// TwinCAT 3 PLC project PLC
// Title: NotificationExample
// Company: Red Rock Controls Limited
// Author: Roger Christopher
// ProjectVersion: 1.0.1.0
// ProgramVersion: 3.1.4024.12
// libraries:
//   Tc2_Standard, * (Beckhoff Automation GmbH)
//   Tc2_System, * (Beckhoff Automation GmbH)
//   Tc3_Module, * (Beckhoff Automation GmbH)
//   tcl_BaseClasses, * (Red Rock Controls Limited)
// project tree:
//   GVLs/ Notifications.TcGVL
//   / PlcTask.TcTTO, PlcTask2.TcTTO
//   POUs/ MAIN_Task1.TcPOU, MAIN_Task2.TcPOU, T_MachineSettingsServer.TcPOU, T_MachineSettingsClient.TcPOU
//   Version/ Global_Version.TcGVL
// real-time tasks:
//   TASK PlcTask1: cycle T#1ms, priority 4, ADS port 350
//   TASK PlcTask2: cycle T#1ms, priority 5, ADS port 351

CONFIGURATION PLC
    RESOURCE PLC ON TwinCAT3
        TASK PlcTask(INTERVAL := T#1ms, PRIORITY := 4);
        TASK PlcTask2(INTERVAL := T#1ms, PRIORITY := 5);
        PROGRAM MAIN_Task1 WITH PlcTask : MAIN_Task1;
        PROGRAM MAIN_Task2 WITH PlcTask2 : MAIN_Task2;
    END_RESOURCE
END_CONFIGURATION

// ---- GVLs/Notifications.TcGVL
{attribute 'qualified_only'}
VAR_GLOBAL
	MachineSettingsLoaded  : T_Notification;
	MachineSettingsUpdated : T_Notification;
END_VAR

// ---- Version/Global_Version.TcGVL
{attribute 'TcGenerated'}
{attribute 'no-analysis'}
{attribute 'linkalways'}
// This function has been automatically generated from the project information.
VAR_GLOBAL CONSTANT
	{attribute 'const_non_replaced'}
	stLibVersion_NotificationExample : ST_LibVersion := (iMajor := 1, iMinor := 0, iBuild := 1, iRevision := 0, nFlags := 0, sVersion := '1.0.1.0');
END_VAR

// ---- POUs/MAIN_Task1.TcPOU
PROGRAM MAIN_Task1
VAR
    MachineSettingsServer : T_MachineSettingsServer; // Sends settings and loaded status to MachineSettingsClient running in separate context (task)
    Init            : BOOL := TRUE;

END_VAR

IF Init THEN
    // Manually resize the args buffer, as resizing 10,000 times produces a very long scan...
    Notifications.MachineSettingsUpdated.Args.Init(StreamLength := 60000);

    // Link the handler to the notification...
    Notifications.MachineSettingsLoaded
        .ClearNotificationHandlers()
    	.AddNotificationHandler(MAIN_Task2.MachineSettingsClient.OnSettingsLoaded);

    Notifications.MachineSettingsUpdated
        .ClearNotificationHandlers()
    	.AddNotificationHandler(MAIN_Task2.MachineSettingsClient.OnSettingsUpdated);

    Init := FALSE;
END_IF

// Run the server...
MachineSettingsServer.CyclicUpdate();

END_PROGRAM

// ---- POUs/T_MachineSettingsServer.TcPOU
FUNCTION_BLOCK T_MachineSettingsServer
VAR
    SettingsLoaded  : BOOL; // raises MachineSettingsLoaded notification, handled by T_MachineSettingsClient
    SettingsUpdated : BOOL; // raises MachoneSettingsUpdated notification, handled by T_MachineSettingsClient

    Settings : ARRAY[1..10000] OF UDINT;

END_VAR

METHOD CyclicUpdate
VAR_INST
    Init     : BOOL := TRUE;
    i        : UDINT;
    SendOnce : BOOL := TRUE; // set true to send single notifications
END_VAR
IF Init THEN
    // clear the flag...
    Init := FALSE;

    // write some values into the settings...
    FOR i := 1 TO 10000 DO
        Settings[i] := i;
    END_FOR
END_IF

IF SettingsLoaded THEN // manually set this flag to send SettingsLoaded notifications...
    IF SendOnce THEN // Set SendOnce to FALSE to send notification every scan - should still work if tasks run on separate isolated cores!
        SettingsLoaded := FALSE; 
    END_IF

    // raise the simple notification with no args...
    Notifications.MachineSettingsLoaded.Raise();
END_IF

IF SettingsUpdated THEN // manually set this flag to send SettingsUpdated notifications...
    IF SendOnce THEN // Set SendOnce to FALSE to send notification every scan - should still work if tasks run on separate isolated cores!
        SettingsUpdated := FALSE; 
    END_IF

    // write the seettings into the notification args...
    FOR i := 1 TO 10000 DO
        Notifications.MachineSettingsUpdated.Args.Add_UDINT(Settings[i]);
    END_FOR

    // raise the notification...
    Notifications.MachineSettingsUpdated.Raise();
END_IF
END_METHOD

END_FUNCTION_BLOCK

// ---- POUs/MAIN_Task2.TcPOU
PROGRAM MAIN_Task2
VAR
	MachineSettingsClient : T_MachineSettingsClient; // Receives settings and loaded status from MachineSettingsServer running in separate context (task)
END_VAR

MachineSettingsClient.HandleNotifications();

END_PROGRAM

// ---- POUs/T_MachineSettingsClient.TcPOU
FUNCTION_BLOCK T_MachineSettingsClient // Handles notifications of settings loaded and settings updated
VAR
    OnSettingsLoaded  : T_NotificationHandler;
    OnSettingsUpdated : T_NotificationHandler;

    SettingsLoadedCount : UDINT;
    LocalSettings       : ARRAY[1..10000] OF UDINT;
END_VAR

METHOD HandleNotifications
VAR
    i                   : UDINT;
END_VAR
IF OnSettingsLoaded.IsRaised() THEN
    // do something...
    SettingsLoadedCount := SettingsLoadedCount + 1;
END_IF

IF OnSettingsUpdated.IsRaised() THEN
    // read the 10,000 settings passed via the notification args...
    FOR i := 1 TO 10000 DO
		// read the arg...
		LocalSettings[i] := OnSettingsUpdated.Args.Read_UDINT();
    END_FOR
END_IF
END_METHOD

END_FUNCTION_BLOCK
